(* CODESYS project PersistantHandler.export

Project tree, tasks and I/O mapping:
  Persistant/
    data type EN_FILE_ERROR
    data type ST_PERSISTANT_VAR
    global variables GVL_PERSISTANT_DATA
    function FC_RESTORE_PERS [ST]
    function FC_SAVE_PERS [ST]
    program PRG_PERSISTANT [ST]
  System Events/
    function SYSEVT_ONLINE_CHANGE [ST]
    function SYSEVT_START [ST]
    function SYSEVT_STOP [ST]
*)

// Persistant/EN_FILE_ERROR
TYPE EN_FILE_ERROR :
(
	UnknownState := 0,
	Busy := 1,
	Done := 2,
	FileCloseError := 4,
	FileWriteError := 5,
	FileReadError := 6,
	FileOpenError := 7
);
END_TYPE

// Persistant/ST_PERSISTANT_VAR
TYPE ST_PERSISTANT_VAR :
STRUCT
	/// Add Retain Vars as used 
	/// NOTE !!! Append a Var only at the End of declaration, 
	/// otherwise the Logfile Crashes !!!
	uiCountOnlineChange		: UINT;	
	uiCountStart			: UINT;
	uiCountStop				: UINT;
	
	// Actual Data
	dYesterday				: DATE;
	
END_STRUCT
END_TYPE

// Persistant/GVL_PERSISTANT_DATA
{attribute 'qualified_only'}
VAR_GLOBAL
	utPersVar	: ST_PERSISTANT_VAR;
END_VAR

// Persistant/FC_RESTORE_PERS
FUNCTION FC_RESTORE_PERS : BYTE
VAR
	bState				: BYTE;
	dwHandler			: RTS_IEC_HANDLE;
	xFileClosedOK		: BOOL;
	lwByteWritten		: lWORD;
	Result				:  RTS_IEC_HANDLE;
	udiResult			: UDINT;
END_VAR
VAR_INPUT
	sFilename	: STRING;
END_VAR
VAR_IN_OUT
	myRetains	: ST_PERSISTANT_VAR;
END_VAR

bState:=1;
dwHandler:=0;
xFileClosedOK:=FALSE;
// Open file
dwHandler:=SysFileOpen(szFile:=GVL_CONFIG.sPersFilename , am:=ACCESS_MODE.AM_READ,pResult := Result );
IF dwHandler > 0 THEN
	// Read file
	lwByteWritten:=SysFileRead(hFile:=dwHandler , pbyBuffer:=ADR(GVL_PERSISTANT_DATA.utPersVar) , ulSize:=SIZEOF(ST_PERSISTANT_VAR),pResult:=Result );
	IF lwByteWritten >0 THEN
		// Close file
		udiResult:=SysFileClose(hFile:=dwHandler);
		IF udiResult = SYS_FILE_STATUS.FS_OK THEN
			bState:=2;
		ELSE
			bState:=4;
		END_IF
	ELSE
		bState:=6;			
	END_IF
ELSE
	bState:=7;	
END_IF

FC_RESTORE_PERS:=bState;

END_FUNCTION

// Persistant/FC_SAVE_PERS
FUNCTION FC_SAVE_PERS : BYTE
VAR
	bState			: BYTE;
	dwHandler		: RTS_IEC_HANDLE;
	xFileClosedOK	: BOOL;
	lwByteWritten	: lWORD;
	Result			: RTS_IEC_HANDLE;
	udiResult			: UDINT;
END_VAR
VAR_INPUT
	sFilename	: STRING;
END_VAR
VAR_IN_OUT
	myRetains	: ST_PERSISTANT_VAR;
END_VAR

bState:=1;
dwHandler:=0;
xFileClosedOK:=FALSE;
// Open file
dwHandler:=SysFileOpen(szFile :=GVL_CONFIG.sPersFilename , am:=ACCESS_MODE.AM_WRITE, pResult := Result  );
IF dwHandler > 0 THEN
	// Write file
	lwByteWritten:=SysFileWrite(hFile:=dwHandler , pbyBuffer:=ADR(GVL_PERSISTANT_DATA.utPersVar) , ulSize:=SIZEOF(ST_PERSISTANT_VAR),pResult:=Result );
	IF lwByteWritten >0 THEN
		// Close file
		udiResult:=SysFileClose(hFile:=dwHandler );
		IF udiResult = SYS_FILE_STATUS.FS_OK  THEN
			bState:=2;
		ELSE
			bState:=4;
		END_IF	
	ELSE
		bState:=5;		
	END_IF	
ELSE
	bState:=7;	
END_IF

FC_SAVE_PERS:=bState;

END_FUNCTION

// Persistant/PRG_PERSISTANT
PROGRAM PRG_PERSISTANT
VAR
		xRestore			: BOOL;
	xSave					: BOOL;
	bSavingState			: EN_FILE_ERROR;
	bRestoringState			: EN_FILE_ERROR;
	///Calc Checksum
	arByte					: ARRAY[0..50] OF BYTE;// Anzahl der Bytes an die Variablenstruktur RetainVar je nach Bedarf anpassen.
	i						: DWORD;
	rChecksum				: REAL;
	rChecksum_old			: REAL;
	dwCountSaveManual		: DWORD;
	dwCountRestoreManual	: DWORD;
END_VAR

//=========================================================
// +++ RESTORE MANUAL +++
//=========================================================
IF xRestore THEN
	xRestore:=FALSE;
	bRestoringState:=FC_RESTORE_PERS(sFilename:=GVL_CONFIG.sPersFilename , myRetains:=GVL_PERSISTANT_DATA.utPersVar );
	dwCountRestoreManual:=dwCountRestoreManual+1;
END_IF

//=========================================================
// +++ SAVE MANUAL +++
//=========================================================
IF xSave THEN
	xSave:=FALSE;
	bSavingState:=FC_SAVE_PERS(sFilename:=GVL_CONFIG.sPersFilename , myRetains:=GVL_PERSISTANT_DATA.utPersVar );
	dwCountSaveManual:=dwCountSaveManual+1;
END_IF

//=========================================================
// +++ CALCULATE CHECKSUM AND AUTO SAVE+++
//=========================================================
MemCopy(pDest:=ADR(arByte) , pSource:=ADR(GVL_PERSISTANT_DATA.utPersVar) , udiSize:=SIZEOF(ST_PERSISTANT_VAR));
rChecksum:=0;
FOR i:=0 TO SIZEOF(ST_PERSISTANT_VAR) BY 1 DO
	rChecksum:=rChecksum + BYTE_TO_REAL(arByte[i])/1000;
END_FOR
IF rChecksum_old <> rChecksum THEN
	xSave:=TRUE;
	rChecksum_old:=rChecksum;
END_IF

END_PROGRAM

// System Events/SYSEVT_ONLINE_CHANGE
FUNCTION SYSEVT_ONLINE_CHANGE : DWORD
VAR_IN_OUT
	EventPrm: CmpApp.EVTPARAM_CmpApp;
END_VAR

// Count lling
GVL_PERSISTANT_DATA.utPersVar.uiCountOnlineChange:=GVL_PERSISTANT_DATA.utPersVar.uiCountOnlineChange+1;
// Do restore
FC_RESTORE_PERS(sFilename:=GVL_CONFIG.sPersFilename , myRetains:=GVL_PERSISTANT_DATA.utPersVar );

END_FUNCTION

// System Events/SYSEVT_START
FUNCTION SYSEVT_START : DWORD
VAR_IN_OUT
	EventPrm: CmpApp.EVTPARAM_CmpApp;
END_VAR
VAR
END_VAR

//Count Calling
GVL_PERSISTANT_DATA.utPersVar.uiCountStart:=GVL_PERSISTANT_DATA.utPersVar.uiCountStart+1;	
// Do restore
FC_RESTORE_PERS(sFilename:=GVL_CONFIG.sPersFilename , myRetains:=GVL_PERSISTANT_DATA.utPersVar );

END_FUNCTION

// System Events/SYSEVT_STOP
FUNCTION SYSEVT_STOP : DWORD
VAR_IN_OUT
	EventPrm: CmpApp.EVTPARAM_CmpAppStop;
END_VAR

// Count Calling
GVL_PERSISTANT_DATA.utPersVar.uiCountStop:=GVL_PERSISTANT_DATA.utPersVar.uiCountStop+1;	
// Do Save
FC_SAVE_PERS(sFilename:=GVL_CONFIG.sPersFilename , myRetains:=GVL_PERSISTANT_DATA.utPersVar );

END_FUNCTION
